FUNCTION_BLOCK RobotinoViewUdp
  (* Standard: 61499-2 *)
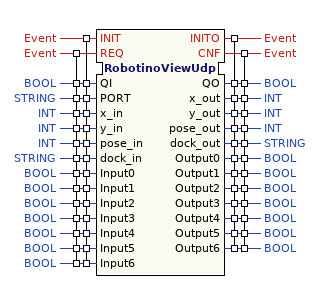
  EVENT_INPUT
    INIT WITH QI, PORT, x_in, y_in, pose_in, dock_in, Input0, Input1, Input2, Input3, Input4, Input5, Input6;
    REQ WITH QI, PORT, x_in, y_in, pose_in, dock_in, Input0, Input1, Input2, Input3, Input4, Input5, Input6;
  END_EVENT
  EVENT_OUTPUT
    INITO WITH QO, x_out, y_out, pose_out, dock_out, Output0, Output1, Output2, Output3, Output4, Output5, Output6;
    CNF WITH QO, x_out, y_out, pose_out, dock_out, Output0, Output1, Output2, Output3, Output4, Output5, Output6;
  END_EVENT
  VAR_INPUT
    QI : BOOL;
    PORT : STRING;
    x_in : INT;
    y_in : INT;
    pose_in : INT;
    dock_in : STRING;
    Input0 : BOOL;
    Input1 : BOOL;
    Input2 : BOOL;
    Input3 : BOOL;
    Input4 : BOOL;
    Input5 : BOOL;
    Input6 : BOOL;
  END_VAR
  VAR_OUTPUT
    QO : BOOL;
    x_out : INT;
    y_out : INT;
    pose_out : INT;
    dock_out : STRING;
    Output0 : BOOL;
    Output1 : BOOL;
    Output2 : BOOL;
    Output3 : BOOL;
    Output4 : BOOL;
    Output5 : BOOL;
    Output6 : BOOL;
  END_VAR
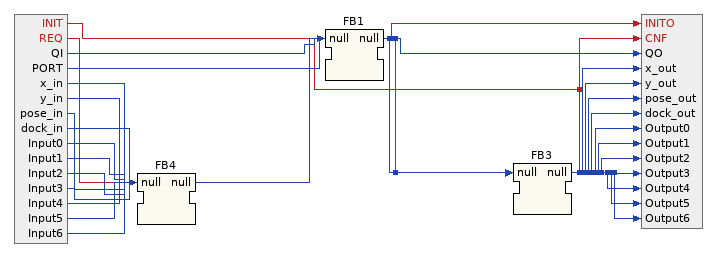
  FBS
    FB1 : ;
    FB3 : ;
    FB4 : ;
  END_FBS
  EVENT_CONNECTIONS
    INIT TO FB1.null;
    FB1.null TO INITO;
    FB1.null TO FB3.null;
    FB3.null TO FB1.null;
    REQ TO FB4.null;
    FB4.null TO FB1.null;
    FB3.null TO CNF;
  END_CONNECTIONS
  DATA_CONNECTIONS
    PORT TO FB1.null;
    QI TO FB1.null;
    FB1.null TO QO;
    FB1.null TO FB3.null;
    FB3.null TO x_out;
    FB3.null TO y_out;
    FB3.null TO pose_out;
    FB3.null TO dock_out;
    FB3.null TO Output0;
    FB3.null TO Output1;
    FB3.null TO Output2;
    FB3.null TO Output3;
    FB3.null TO Output4;
    FB3.null TO Output5;
    FB3.null TO Output6;
    x_in TO FB4.null;
    y_in TO FB4.null;
    pose_in TO FB4.null;
    dock_in TO FB4.null;
    Input0 TO FB4.null;
    Input1 TO FB4.null;
    Input2 TO FB4.null;
    Input3 TO FB4.null;
    Input4 TO FB4.null;
    Input5 TO FB4.null;
    Input6 TO FB4.null;
    FB4.null TO FB1.null;
  END_CONNECTIONS
END_FUNCTION_BLOCK
